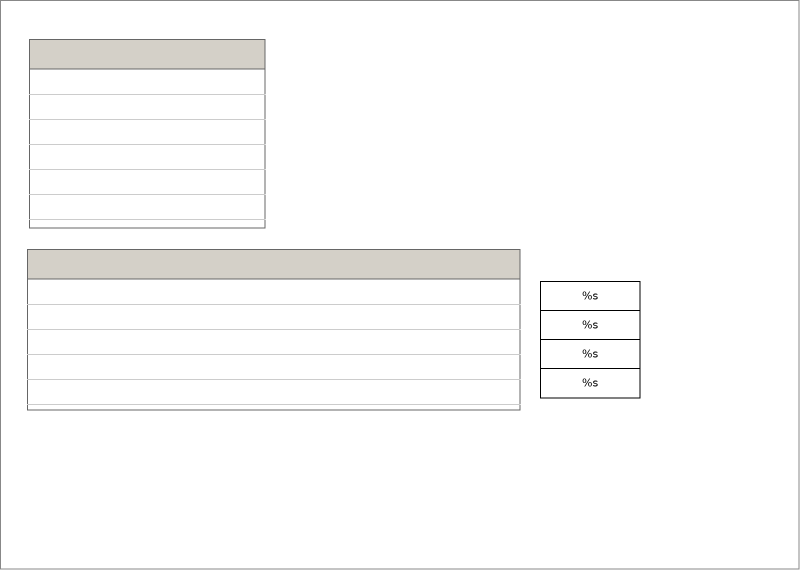
VISUALIZATION VIS_FootPedal  // 800x570
    Table (29,39 236x189), data array: stInput.biFootPedal
        p3854506369: stInput.biFootPedal[INDEX].PedalPressed1
        p1892666644: stInput.biFootPedal[INDEX].PedalPressed2
        p338671338: stInput.biFootPedal[INDEX].PedalPressed3
        Columns.Column.[2].Template: toggle stInput.biFootPedal[INDEX].PedalPressed3
        Columns.Column.[0].Template: toggle stInput.biFootPedal[INDEX].PedalPressed1
        Columns.Column.[1].Template: toggle stInput.biFootPedal[INDEX].PedalPressed2
    Table (27,249 493x161), data array: GVL_API.stFootPedal
        p1218418051: P_FootPedal.FB_FootPedal[INDEX].state
        p746581629: P_FootPedal.FB_FootPedal[INDEX].pressed
        p3104783080: P_FootPedal.FB_FootPedal[INDEX].ton1
        p2501879983: P_FootPedal.FB_FootPedal[INDEX].step
        p7306298: P_FootPedal.FB_FootPedal[INDEX].Reset
        p3854506369: GVL_API.stFootPedal[INDEX].error_code
        p1892666644: GVL_API.stFootPedal[INDEX].state
        p338671338: GVL_API.stFootPedal[INDEX].pressed
        p2170511999: GVL_API.stFootPedal[INDEX].Reset
        p3723444502: GVL_API.stFootPedal[INDEX].debounce_time
        Columns.Column.[4].Template: OnMouseDown: write GVL_API.stFootPedal[INDEX].debounce_time via Default
        Columns.Column.[3].Template: toggle GVL_API.stFootPedal[INDEX].Reset
    Rectangle (540,281 100x30), "%s", text variable: P_FootPedal.FB_FootPedal[1].ton1.ET
    Rectangle (540,310 100x30), "%s", text variable: P_FootPedal.FB_FootPedal[2].ton1.ET
    Rectangle (540,339 100x30), "%s", text variable: P_FootPedal.FB_FootPedal[3].ton1.ET
    Rectangle (540,368 100x30), "%s", text variable: P_FootPedal.FB_FootPedal[4].ton1.ET
END_VISUALIZATION

(* stored: Version 1.1.0.1, ProductVersion 3.1.4024.11
   Visu VIS_FootPedal: Id {147c0b6f-c0b3-4524-8489-346a3352b1d9} *)
